ABB RobotStudio station: Solution4_1_20180324-193448.rsstn

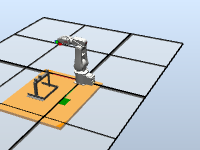
Station Solution4_1 (saved by RobotStudio 6.6.7701.1025)
Controller IRB_120_3kg_0.58m
  mechanical unit ROB_1: IRB120_3_58__01, 6 joints, base frame (0, 0, 0) mm
Layout (positions relative to the parent item):
  - IRB120_3_58__01 [mechanism, from Robots\IRB120_3_58_G_01.rslib] at (0, 0, 0) mm; joint values [0, 0, 0, 0, 0.5236, 0] (rad or m)
  - shelf_2 [part] at (500, 700, 0) mm, rotated rx 90 ry 0 rz -90 deg
  - table [part] at (-300, -100, 0) mm, rotated rx -90 ry 0 rz 0 deg
  - ciruit [part] at (-100, 500, 0) mm, rotated rx 90 ry 0 rz 90 deg
